// TIA Portal V16 export
// export: Created 2022-07-21T09:35:16.4566816Z, ExportSetting WithDefaults, DisplayName Totally Integrated Automation Portal, DisplayVersion V16 Update 4, DisplayName TIA Portal Version Control Interface, DisplayVersion V16 Update 2, DisplayName TIA Portal Openness, DisplayVersion V16 Update 4, DisplayName SINAMICS Startdrive Advanced, DisplayVersion V16 Update 5, DisplayName SINAMICS Startdrive G130, G150, S120, S150, SINAMICS MV, S210, DisplayVersion V16 Update 5, DisplayName SINAMICS Startdrive G110M, G120, G120C, G120D, G120P, G115D, DisplayVersion V16 Update 5, DisplayName STEP 7 Professional, DisplayVersion V16 Update 4, DisplayName STEP 7 Safety, DisplayVersion V16, DisplayName WinCC Advanced, DisplayVersion V16 Update 4
FUNCTION_BLOCK "fbReadingWindow"   // FB86, LAD
TITLE = Read window / Okno odczytu
{ S7_Optimized_Access := 'TRUE' }
VERSION : 0.1
// inTrigger : set continous signal, e.g. transport through sensor. If signal is too short (e.g. edge detection) then set TriggerExtension to e.g. 500ms / inTrigger : ustawić sygnał ciągły, np. przejazd przez czujnik. Jeżeli zbocze to ustawić TriggerExtension, np. 500ms
// stored: AutoNumber true, IsIECCheckEnabled true, IsRetainMemResEnabled false, MemoryReserve 100, SetENOAutomatically false, UDAEnableTagReadback false
   VAR_INPUT
      inTrigger { ExternalAccessible := 'False'; ExternalVisible := 'False'; ExternalWritable := 'False'} : Bool;   // Trigger
      inTriggerExtension { ExternalAccessible := 'False'; ExternalVisible := 'False'; ExternalWritable := 'False'} : Time;   // Wydłużenie sygnału trigger / Extend trigger signal
      inTimeoutNoData { ExternalAccessible := 'False'; ExternalVisible := 'False'; ExternalWritable := 'False'} : Time;   // Czas na do wygenerowania sygnału braku danych / Timeout "no data"
      inDataReceived { ExternalAccessible := 'False'; ExternalVisible := 'False'; ExternalWritable := 'False'} : Bool;   // Nowe dane z kamery / New data from camera
   END_VAR
   VAR_OUTPUT
      ouWaitingForData { ExternalAccessible := 'False'; ExternalVisible := 'False'; ExternalWritable := 'False'} : Bool;   // Oczekiwanie na nowy telegram / Wait for new telegram
      ouReqTrigger { ExternalAccessible := 'False'; ExternalVisible := 'False'; ExternalWritable := 'False'} : Bool;   // Żądanie wyzwolenia kamery / Camera trigger request
   END_VAR
   VAR
      sUsedTriggerExtension { ExternalAccessible := 'False'; ExternalVisible := 'False'; ExternalWritable := 'False'} : Time;
      sUsedTimeoutNoData { ExternalAccessible := 'False'; ExternalVisible := 'False'; ExternalWritable := 'False'} : Time;
      sREReqTrigger { ExternalAccessible := 'False'; ExternalVisible := 'False'; ExternalWritable := 'False'} : Bool;
      sFEReqTrigger { ExternalAccessible := 'False'; ExternalVisible := 'False'; ExternalWritable := 'False'} : Bool;
      sRETrigger { ExternalAccessible := 'False'; ExternalVisible := 'False'; ExternalWritable := 'False'} : Bool;
      sFETrigger { ExternalAccessible := 'False'; ExternalVisible := 'False'; ExternalWritable := 'False'} : Bool;
      sTONTimeOutNoData { S7_SetPoint := 'True'} : TON_TIME;
      sTONTriggerExtension { S7_SetPoint := 'True'} : TON_TIME;
   END_VAR
   VAR_TEMP
      tREReqTrigger : Bool;
      tFEReqTrigger : Bool;
      tRETrigger : Bool;
      tFETrigger : Bool;
   END_VAR
   VAR_TEMP   // added for the SCL form of the ladder/FBD networks
      _w1 : Bool;
      _w2 : Bool;
      _w3 : Bool;
      _w4 : Bool;
   END_VAR
BEGIN

REGION Network 1: Extend trigger signal / Wydłużenie sygnału wyzwolenia
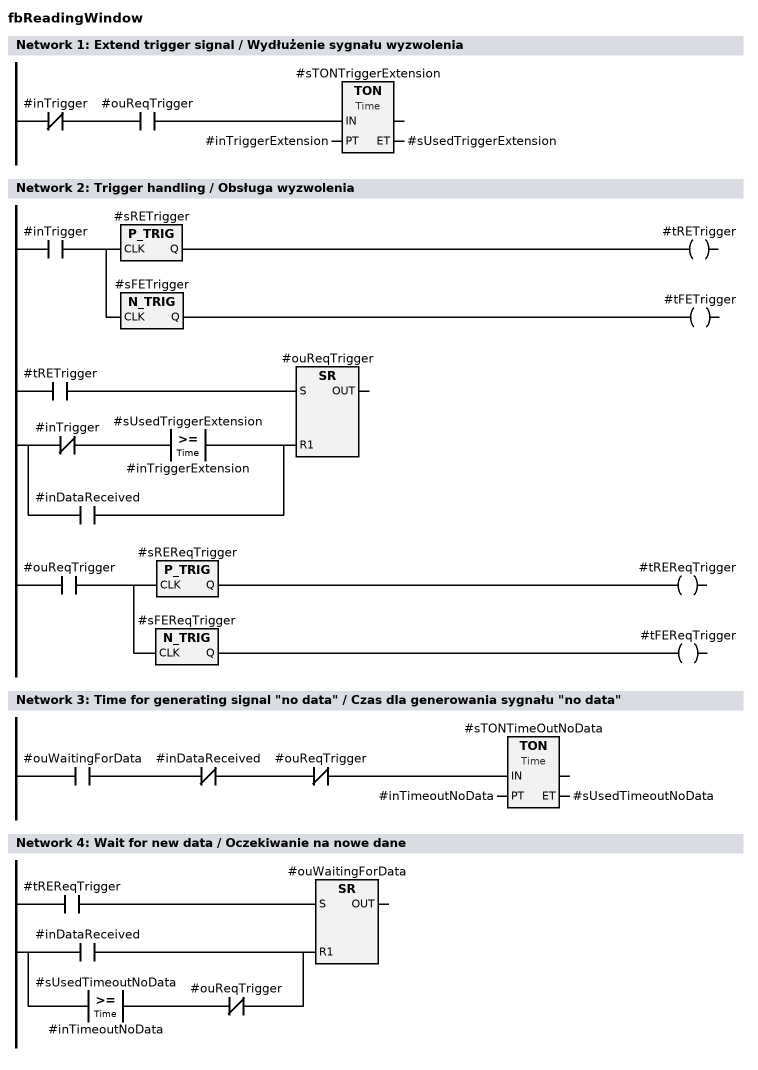
   RUNG wire#powerrail
      I_Contact( #inTrigger )
      Contact( #ouReqTrigger )
      { S7_Templates := "time_type := Time" } #sTONTriggerExtension.TON(pt := #inTriggerExtension, et => #sUsedTriggerExtension)
   END_RUNG
   // the same network as SCL:
   #sTONTriggerExtension(IN := NOT #inTrigger AND #ouReqTrigger,   // TON
                         PT := #inTriggerExtension,
                         ET => #sUsedTriggerExtension);
END_REGION

REGION Network 2: Trigger handling / Obsługa wyzwolenia
   RUNG wire#powerrail
      Contact( #inTrigger )
      wire#w1
      P_Trig( #sRETrigger )
      Coil( #tRETrigger )
   END_RUNG
   RUNG wire#w1
      N_Trig( #sFETrigger )
      Coil( #tFETrigger )
   END_RUNG
   RUNG wire#powerrail
      Contact( #tRETrigger )
      S_SR(operand := #ouReqTrigger, r1 := wire#w2)
   END_RUNG
   RUNG wire#powerrail
      I_Contact( #inTrigger )
      { S7_Templates := "SrcType := Time" } GE_Contact(in1 := #sUsedTriggerExtension, in2 := #inTriggerExtension)
   END_RUNG wire#w2
   RUNG wire#powerrail
      Contact( #inDataReceived )
   END_RUNG wire#w2
   RUNG wire#powerrail
      Contact( #ouReqTrigger )
      wire#w3
      P_Trig( #sREReqTrigger )
      Coil( #tREReqTrigger )
   END_RUNG
   RUNG wire#w3
      N_Trig( #sFEReqTrigger )
      Coil( #tFEReqTrigger )
   END_RUNG
   // the same network as SCL:
   #_w1 := #inTrigger AND NOT #sRETrigger;   // rising edge
   #sRETrigger := #inTrigger;
   #tRETrigger := #_w1;
   #_w2 := NOT #inTrigger AND #sFETrigger;   // falling edge
   #sFETrigger := #inTrigger;
   #tFETrigger := #_w2;
   IF #tRETrigger THEN
       #ouReqTrigger := TRUE;   // SR flip-flop
   END_IF;
   IF (NOT #inTrigger AND (#sUsedTriggerExtension >= #inTriggerExtension)) OR #inDataReceived THEN
       #ouReqTrigger := FALSE;
   END_IF;
   #_w3 := #ouReqTrigger AND NOT #sREReqTrigger;   // rising edge
   #sREReqTrigger := #ouReqTrigger;
   #tREReqTrigger := #_w3;
   #_w4 := NOT #ouReqTrigger AND #sFEReqTrigger;   // falling edge
   #sFEReqTrigger := #ouReqTrigger;
   #tFEReqTrigger := #_w4;
END_REGION

REGION Network 3: Time for generating signal "no data" / Czas dla generowania sygnału "no data"
   RUNG wire#powerrail
      Contact( #ouWaitingForData )
      I_Contact( #inDataReceived )
      I_Contact( #ouReqTrigger )
      { S7_Templates := "time_type := Time" } #sTONTimeOutNoData.TON(pt := #inTimeoutNoData, et => #sUsedTimeoutNoData)
   END_RUNG
   // the same network as SCL:
   #sTONTimeOutNoData(IN := #ouWaitingForData AND NOT #inDataReceived AND NOT #ouReqTrigger,   // TON
                      PT := #inTimeoutNoData,
                      ET => #sUsedTimeoutNoData);
END_REGION

REGION Network 4: Wait for new data / Oczekiwanie na nowe dane
   RUNG wire#powerrail
      Contact( #tREReqTrigger )
      S_SR(operand := #ouWaitingForData, r1 := wire#w1)
   END_RUNG
   RUNG wire#powerrail
      Contact( #inDataReceived )
   END_RUNG wire#w1
   RUNG wire#powerrail
      { S7_Templates := "SrcType := Time" } GE_Contact(in1 := #sUsedTimeoutNoData, in2 := #inTimeoutNoData)
      I_Contact( #ouReqTrigger )
   END_RUNG wire#w1
   // the same network as SCL:
   IF #tREReqTrigger THEN
       #ouWaitingForData := TRUE;   // SR flip-flop
   END_IF;
   IF #inDataReceived OR ((#sUsedTimeoutNoData >= #inTimeoutNoData) AND NOT #ouReqTrigger) THEN
       #ouWaitingForData := FALSE;
   END_IF;
END_REGION
END_FUNCTION_BLOCK
